FUNCTION_BLOCK FB_Cycle IMPLEMENTS I_Cycle
VAR_INPUT
END_VAR
VAR_OUTPUT
END_VAR
VAR
END_VAR

METHOD PUBLIC M_Cycle
VAR_INPUT
END_VAR
END_METHOD

END_FUNCTION_BLOCK

(* stored: Version 1.1.0.1
   POU FB_Cycle: Id {e74cce6f-550c-444b-8cdf-19b824901777}, SpecialFunc None
   Method M_Cycle: Id {c23b40fd-4755-4d58-9e6c-63dc34a4b87e} *)
